// TIA Portal project "Project15" (V15.1)

(* hardware
DEVICE "S7-1200 station_1"  S7-1200 Station
   slot 0: "Rack_0"  S7-1200 Rack  Rack  V1.0
   slot 1: "PLC_1"  CPU 1214C AC/DC/Rly  6ES7 214-1BG40-0XB0  V4.2
*)

// ===== PLC "PLC_1"  CPU 1214C AC/DC/Rly =====

VAR_GLOBAL   // PLC tag table "Default tag table"
   "start" AT %I0.0 : Bool;
   "sistem start" AT %M0.1 : Bool;
   "stop" AT %I0.2 : Bool;
   "zaman" AT %MD50 : Time;
   "motor1" AT %Q54.0 : Bool;
   "motor2" AT %Q58.0 : Bool;
   "başa al" AT %M62.0 : Bool;
   "başa al2" AT %M62.1 : Bool;
END_VAR

// folder: System blocks/Program resources

DATA_BLOCK "Timer1"   // DB1
{ S7_Optimized_Access := 'TRUE' }
AUTHOR : Simatic
FAMILY : IEC
NAME : IEC_TMR
VERSION : 1.0
// stored: InstanceOfName IEC_TIMER
"IEC_TIMER"
BEGIN
END_DATA_BLOCK

// folder: (top level)

ORGANIZATION_BLOCK "Main"   // OB1, LAD, ProgramCycle
TITLE = "Main Program Sweep (Cycle)"
{ S7_Optimized_Access := 'TRUE' }
VERSION : 0.1
   VAR_INPUT
      Initial_Call : Bool;   // Initial call of this OB
      Remanence : Bool;   // =True, if remanent data are available
   END_VAR
BEGIN

REGION Network 1
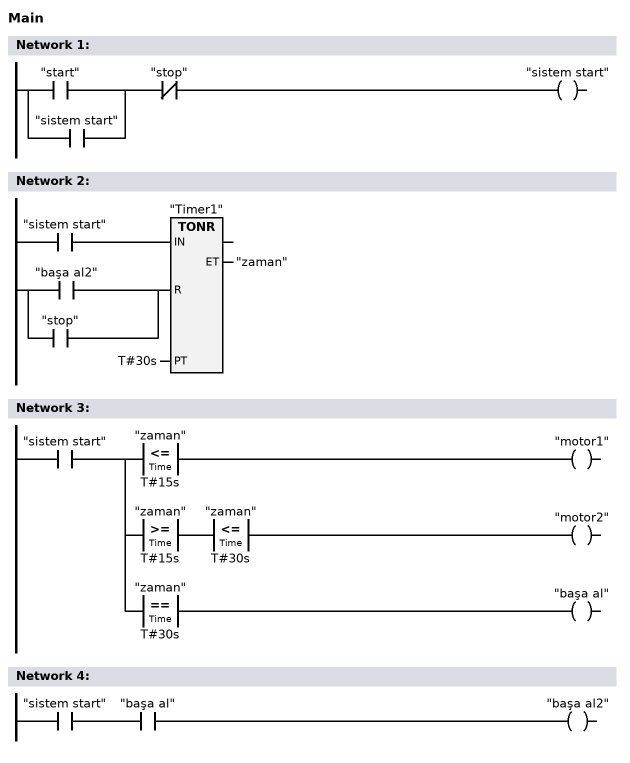
   RUNG wire#powerrail
      Contact( "start" )
      wire#w1
      I_Contact( "stop" )
      Coil( "sistem start" )
   END_RUNG
   RUNG wire#powerrail
      Contact( "sistem start" )
   END_RUNG wire#w1
   // the same network as SCL:
   "sistem start" := ("start" OR "sistem start") AND NOT "stop";
END_REGION

REGION Network 2
   "Timer1".TONR(IN := "sistem start", R := "başa al2" OR "stop", PT := T#30s, ET => "zaman");
END_REGION

REGION Network 3
   RUNG wire#powerrail
      Contact( "sistem start" )
      wire#w1
      { S7_Templates := "SrcType := Time" } LE_Contact(in1 := "zaman", in2 := T#15s)
      Coil( "motor1" )
   END_RUNG
   RUNG wire#w1
      { S7_Templates := "SrcType := Time" } GE_Contact(in1 := "zaman", in2 := T#15s)
      { S7_Templates := "SrcType := Time" } LE_Contact(in1 := "zaman", in2 := T#30s)
      Coil( "motor2" )
   END_RUNG
   RUNG wire#w1
      { S7_Templates := "SrcType := Time" } EQ_Contact(in1 := "zaman", in2 := T#30s)
      Coil( "başa al" )
   END_RUNG
   // the same network as SCL:
   "motor1" := "sistem start" AND ("zaman" <= T#15s);
   "motor2" := "sistem start" AND ("zaman" >= T#15s) AND ("zaman" <= T#30s);
   "başa al" := "sistem start" AND ("zaman" = T#30s);
END_REGION

REGION Network 4
   RUNG wire#powerrail
      Contact( "sistem start" )
      Contact( "başa al" )
      Coil( "başa al2" )
   END_RUNG
   // the same network as SCL:
   "başa al2" := "sistem start" AND "başa al";
END_REGION
END_ORGANIZATION_BLOCK